{attribute 'GeneratedUsingTerminal: EK1100-0000-0018'}
{attribute addProperty BoxType "EK1100-0000-0018"}
{attribute addProperty Id "A_0017_BK1250_0000_0018A_0017_BK1250_0000_0018_8BB339150"}
{attribute addProperty CRC "4252368664"}
{attribute addProperty Size "0"}
TYPE Term_21_EK1100_FD75FF18 EXTENDS EK1100_1FC0878B :
STRUCT
	{attribute addProperty Name "A_0017_BK1250_0000_0018"}
	{attribute addProperty PreviousPort "Term 21 (EK1100) : B"}
	A_0017_BK1250_0000_0018 : A_0017_BK1250_0000_0018_8BB33915;
END_STRUCT
END_TYPE

(* stored: Version 1.2.0.0, ProductVersion 3.1.4024.9
   DUT Term_21_EK1100_FD75FF18: Id {b372b5b9-3f09-4ee2-adee-836a552a963d} *)
